Omron CX-Programmer project 新工程 (CX-Programmer 9.73)

# PLC 新PLC1: CJ1M CPU11

## Global symbols (name address type ; comment)
2000 CHANNEL  ; 打螺丝个数显示
2000.01 BOOL  ; 参数1
2000.02 BOOL  ; 参数2
2000.03 BOOL  ; DRIVER PROGRAM CH3
2000.04 BOOL  ; DRIVER PROGRAM CH4
2000.07 BOOL  ; BZ
2000.08 BOOL  ; 正常指示
2000.09 BOOL  ; 异常指示
2000.10 BOOL  ; OK
2000.11 BOOL  ; NG指示
2000.12 BOOL  ; BZ
2006.00 BOOL  ; 前A2吐油SOL
2006.02 BOOL  ; 前A1吐油SOL
2006.04 BOOL  ; A1后吐油
2006.06 BOOL  ; A2后吐油
2006.08 BOOL  ; 打油SOL
2007.00 BOOL  ; 涂布运转准备条件
2007.01 BOOL  ; MS运转准备条件
2007.06 BOOL  ; 第一步OK
2007.07 BOOL  ; 第二步OK
2007.08 BOOL  ; 第三步OK
2007.09 BOOL  ; 第四步OK
2007.11 BOOL  ; 不良
2007.12 BOOL  ; 蜂鸣器
2008.00 BOOL  ; 工件确认
2008.01 BOOL  ; 组装可信号
2008.02 BOOL  ; 完了信号
2008.03 BOOL  ; 完了信號
2008.04 BOOL  ; 报警信号
2008.05 BOOL  ; 打螺丝手柄开关
2008.08 BOOL  ; 组装回数选择
2008.09 BOOL  ; 不良解除
2008.10 BOOL  ; 消音
2008.15 BOOL  ; 运转准备ON
2014.00 BOOL  ; 前有工件传感器
2014.01 BOOL  ; 前吐油传感器
2014.02 BOOL  ; 后有工件传感器
2014.03 BOOL  ; 后吐油传感器
2014.04 BOOL  ; 后吐油开始传感器
2014.05 BOOL  ; 前吐油开始传感器
2014.06 BOOL  ; GREASE COATING CONF.2R
2014.07 BOOL  ; GREASE COATING CONF.2L
2014.08 BOOL  ; WORKPIECE CONFIEMATION
2014.09 BOOL  ; WORKPIECE SET MEMORY
2015.00 BOOL  ; 运转准备ON
2015.03 BOOL  ; 非常停止
2015.05 BOOL  ; -
2015.06 BOOL  ; 自动
2015.07 BOOL  ; 不良解除
2015.08 BOOL  ; 消音
2015.09 BOOL  ; 后涂布手动
2015.10 BOOL  ; 前涂布手动
2015.15 BOOL  ; 獶盽氨ゎ
2100.00 BOOL  ; WORKPIECE SET MEMORY
253.08 BOOL  ; CPU BATTERY LOWER
3000.00 BOOL  ; AUTO. RUN
3000.01 BOOL  ; START
3200.00 BOOL  ; PC FAULT
3200.01 BOOL  ; PATTERN FAULT
3200.02 BOOL  ; CYCLE TIME  OVER
3200.04 BOOL  ; GREASE COATING FAULT
3200.05 BOOL  ; GREASE COATING CONF. SENSOR FAULT
3201.00 BOOL  ; FAULT
3201.01 BOOL  ; ALARM RESET
3201.03 BOOL  ; FAULT RESET
3210.00 BOOL  ; RESTART PROTECTION
3210.01 BOOL  ; CONDITION OF AUTO RUN
3210.15 BOOL  ; CYCLE COMPLETE
3211.00 BOOL  ; INDIV. STEP UP
3211.04 BOOL  ; STEP UP
3211.06 BOOL  ; AUTO. RUN (DIFU)
3211.08 BOOL  ; NOT STEP MOTION
3220.00 BOOL  ; GREASE COATING START:1R
3220.01 BOOL  ; GREASE COATING GOOD:1R
3220.02 BOOL  ; GREASE COATING FAULT:1R
3221.00 BOOL  ; GREASE COATING START:1L
3221.01 BOOL  ; GREASE COATING GOOD:1L
3221.02 BOOL  ; GREASE COATING FAULT:1L
3222.00 BOOL  ; GREASE COATING START:2R
3222.01 BOOL  ; GREASE COATING GOOD:2R
3222.02 BOOL  ; GREASE COATING FAULT:2R
3223.00 BOOL  ; GREASE COATING START:2L
3223.01 BOOL  ; GREASE COATING GOOD:2L
3223.02 BOOL  ; GREASE COATING FAULT:2L
3223.08 BOOL  ; AIR SUPPLY ON
3230.00 BOOL  ; �幡R猳
3230.01 BOOL  ; GREASE COATING 1SHOT:1L
3230.02 BOOL  ; GREASE COATING 1SHOT:2R
3230.03 BOOL  ; GREASE COATING 1SHOT:2L
3240.00 BOOL  ; PATTERN FAULT
3250.00 BOOL  ; 後吐油非
3260.01 BOOL  ; spare
3260.02 BOOL  ; spare
32.00 BOOL  ; 放工件脉冲
32.01 BOOL  ; CYCLE开始
32.02 BOOL  ; NG
32.03 BOOL  ; 手动打螺丝PLS
32.04 BOOL  ; 初始化完成信号
33.00 BOOL  ; 驱动器开始控制
33.01 BOOL  ; 1st. COMPLETE BZ
33.02 BOOL  ; 2nd. COMPLETE BZ
33.03 BOOL  ; 固定过程完成
33.04 BOOL  ; 步完成蜂鸣器叫
33.05 BOOL  ; 2过程完成蜂鸣器
33.06 BOOL  ; 步完成蜂鸣器
33.07 BOOL  ; OK
33.08 BOOL  ; NG
33.09 BOOL  ; NG RESET
33.10 BOOL  ; NG
33.11 BOOL  ; BZ复位
33.12 BOOL  ; BZ
33.13 BOOL  ; 3nd. COMPLETE BZ
34.00 BOOL  ; 机种选择2
34.01 BOOL  ; 机种选择1
50.00 BOOL  ; A1后吐油
50.01 BOOL  ; 第一步后吐油完成
50.02 BOOL  ; A1前吐油
50.03 BOOL  ; 第二步前吐油完成
50.05 BOOL  ; 第三步后吐油完成
50.06 BOOL  ; A1后吐油
50.07 BOOL  ; 第四部后吐油完成
51.00 BOOL  ; 产品确认
51.02 BOOL  ; 报警
52.00 BOOL  ; A2后吐油
52.01 BOOL  ; A2后吐油
52.02 BOOL  ; A2前吐油
52.03 BOOL  ; A2前吐油
52.04 BOOL  ; A1后吐油
52.05 BOOL  ; A2后吐油
52.06 BOOL  ; A2后吐油
52.07 BOOL  ; A2后吐油
52.08 BOOL  ; A2后吐油
53.00 BOOL  ; 后吐油无工件确认
55.00 BOOL  ; 下一步吐油可以
55.01 BOOL  ; 第三步前吐油条件
58.09 BOOL  ; OK
59.00 BOOL  ; 工件正常完成
6014.00 BOOL  ; DUMMY
60.00 BOOL  ; 工件非正常移開
60.01 BOOL  ; 工件非正常移開
60.02 BOOL  ; 故障周期復位
60.03 BOOL  ; NG
60.04 BOOL  ; NG
68.00 BOOL  ; 复位OK
68.01 BOOL  ; 复位OK
80.00 BOOL  ; 自动停止PLS
80.01 BOOL  ; 一次吐油完了
80.02 BOOL  ; 吐油之後拿掉工件
80.03 BOOL  ; �R猳ok
80.04 BOOL  ; 吐油ok後拿掉工件
81.00 BOOL  ; �幡R猳
81.01 BOOL  ; 一次吐油完了
81.02 BOOL  ; 吐油之後拿掉工件
81.03 BOOL  ; �R猳ok
81.04 BOOL  ; 吐油ok後拿掉工件
82.00 BOOL  ; 手动前涂布
82.01 BOOL  ; 手动后涂布
83.00 BOOL  ; NG
83.01 BOOL  ; 蜂鸣器
90.00 BOOL  ; OK RESET START READY
90.01 BOOL  ; OK RESTART
98.00 BOOL  ; COUNTER RESET PLS
A395.11 BOOL  ; Flash MEMORY FAULT
C0118 BOOL  ; 前吐油計數
C0205 BOOL  ; 后涂布计数
D10 CHANNEL  ; 打螺丝个数
D200 CHANNEL  ; 前注油周期
D210 CHANNEL  ; 后注油周期
D220 CHANNEL  ; 注油顺序
D280 CHANNEL  ; 总生产数
H0.00 BOOL  ; Step_0丂
H0.01 BOOL  ; Step_1
H0.02 BOOL  ; Step_2
H0.03 BOOL  ; Step_3
H0.04 BOOL  ; Step_4
H0.05 BOOL  ; Step_5
H0.06 BOOL  ; Step_6
H0.07 BOOL  ; Step_7
H10 CHANNEL  ; BIT SHIFT REGISTER
H10.00 BOOL  ; 初始工作时接通
H10.01 BOOL  ; 1st. TORQUE UP
H10.02 BOOL  ; 2nd. TORQUE UP
H10.03 BOOL  ; 3rd. TORQUE UP
H1.00 BOOL  ; Step_0
H1.01 BOOL  ; Step_1
H1.02 BOOL  ; Step_2
H1.03 BOOL  ; Step_3
H1.04 BOOL  ; Step_4
T0008 BOOL  ; CYCLE TIME
T0010 BOOL  ; 自動延時
T0011 BOOL  ; INDIV. MODE
T0018 BOOL  ; OK
T0020 BOOL  ; WORKPIECE CONF. TIMER :1R
T0021 BOOL  ; WORKPIECE CONF. TIMER :1L
T0030 BOOL  ; WORKPIECE CONF. TIMER :2R
T0031 BOOL  ; WORKPIECE CONF. TIMER :2L
T0060 BOOL  ; GREASE COATING TIME:1R
T0061 BOOL  ; GREASE COATING TIME:1L
T0062 BOOL  ; GREASE COATING TIME:2R
T0063 BOOL  ; GREASE COATING TIME:2L
T0100 BOOL  ; 前有工件延时
T0101 BOOL  ; 前吐油延时
T0102 BOOL  ; 后有工件延时
T0103 BOOL  ; 后吐油延时
T0104 BOOL  ; GREASE COATING CONFIRMATION:1R
T0105 BOOL  ; GREASE COATING CONFIRMATION:1L
T0106 BOOL  ; GREASE COATING CONFIRMATION:2R
T0107 BOOL  ; GREASE COATING CONFIRMATION:2L
T0108 BOOL  ; WORKPIECE CONFIRMATION
T0109 BOOL  ; NON WORKPIECE CONFIRMATION
T0110 BOOL  ; 后吐油开始延时
T0111 BOOL  ; 前吐油开始延时
T0112 BOOL  ; 前涂布手动延时
T0113 BOOL  ; 后涂布手动延时
T0114 BOOL  ; 运转准备输入延时
T0115 BOOL  ; 自动延时
T0119 BOOL  ; 前拿掉工件后延时
T0121 BOOL  ; 后拿掉工件后延时
T0131 BOOL  ; 工件检知延时
T0132 BOOL  ; A1A2后吐油时间
T0133 BOOL  ; A1A2前吐油时间
T0135 BOOL  ; A1A2后吐油时间
T0140 BOOL  ; 工件检知无延时
T0142 BOOL  ; 工件检知无RESET
T0150 BOOL  ; A1后吐油时间
T0151 BOOL  ; A2后吐油时间
T0152 BOOL  ; A1前吐油时间
T0153 BOOL  ; A2前吐油时间
T0154 BOOL  ; A1A2后吐油时间
T0155 BOOL  ; A1吐油时间
T0156 BOOL  ; A2后吐油时间
T0157 BOOL  ; 后油油无检知工件延时
T0158 BOOL  ; A1后吐油时间
T0159 BOOL  ; A2后吐油时间
T0200 BOOL  ; 工件确认延时
T0201 BOOL  ; 工件移开时间
T0202 BOOL  ; 手动打螺丝延时
T0203 BOOL  ; 完了信号延时
T0204 BOOL  ; 驱动器开始信号延时
T0211 BOOL  ; 1st完成BZ Time
T0212 BOOL  ; 2nd完成 BZ Time
T0213 BOOL  ; 3nd完成BZTime
T0214 BOOL  ; 1固定完成时间
T0215 BOOL  ; 2固定完成时间
T0216 BOOL  ; 1固定完成时间
T0221 BOOL  ; 工件移开短延时
T0222 BOOL  ; 蜂鸣器叫时间
T0230 BOOL  ; 第1步完成响时间
T0231 BOOL  ; 第2步完成响时间
T0232 BOOL  ; 第3步完成响时间
T0233 BOOL  ; 第5步完成响时间
T0300 BOOL  ; 前A1 ON持续时间
T0301 BOOL  ; 前A2 ON开始时间
T0302 BOOL  ; 前A2 ON持续时间
T0303 BOOL  ; 前注油CYCLE结束
T0310 BOOL  ; 后A1 ON持续时间
T0311 BOOL  ; 后A2 ON开始时间
T0312 BOOL  ; 后A2 ON持续时间
T0313 BOOL  ; 后注油CYCLE结束
T10 CHANNEL  ; AUTO. MODE
T11 CHANNEL  ; INDIV. MODE
T20 CHANNEL  ; WORKPIECE CONF. TIMER :1R
T21 CHANNEL  ; WORKPIECE CONF. TIMER :1L
T30 CHANNEL  ; WORKPIECE CONF. TIMER :2R
T31 CHANNEL  ; WORKPIECE CONF. TIMER :2L
T8 CHANNEL  ; CYCLE TIME
W100.00 BOOL  ; 吐油ON开始打油
W100.01 BOOL  ; 吐油ON开始打油
W200.00 BOOL  ; 前注油 CYCLE 开始
W200.01 BOOL  ; 前A1 ON 辅助
W200.02 BOOL  ; 前A2 ON 辅助
W200.03 BOOL  ; 前吐油确认
W200.04 BOOL  ; 前吐油完成
W200.05 BOOL  ; 前A2 ON开始时间
W200.06 BOOL  ; 前注油CYCLEEND
W210.00 BOOL  ; 后注油 CYCLE 开始
W210.01 BOOL  ; 后A1 ON 辅助
W210.02 BOOL  ; 后A2 ON 辅助
W210.03 BOOL  ; 后吐油确认
W210.04 BOOL  ; 2部吐油完成
W210.05 BOOL  ; 后A2 ON开始时间
W210.06 BOOL  ; 后注油CYCLEEND
W220.00 BOOL  ; 第一步OK
W220.01 BOOL  ; 第二步OK
W220.02 BOOL  ; 第三步OK
W220.03 BOOL  ; 第四步OK
W230.00 BOOL  ; 第1步完成响一声
W231.01 BOOL  ; 第2步完成响一声
W231.02 BOOL  ; 第4步完成响一声
W231.03 BOOL  ; 第4步完成响一声
W27.04 BOOL  ; 完成蜂鸣器叫一声
W50.07 BOOL  ; 急停报警
W50.08 BOOL  ; 急停蜂鸣器
TUYOU 功能块1
后吐油 功能块1
前吐油 功能块1
吐油 功能块1
吐油1 功能块1
Further comments
1 |  | 2000.00 | c4ded7b2cadebdc0b0c42028c8bcde92f782df29 | 20
2 |  | 2000.01 | c4ded7b2cadeccdfdbb8ded7d120434831 | b2cecafd31
3 |  | 2000.02 | c4ded7b2cadeccdfdbb8ded7d120434832 | b2cecafd32
4 |  | 2000.03 | c4ded7b2cadeccdfdbb8ded7d120434833 | 4452495645522050524f4752414d20434833
5 |  | 2000.04 | c4ded7b2cadeccdfdbb8ded7d120434834 | 4452495645522050524f4752414d20434834
7 |  | 2000.08 | c4ded7b2cade90b38fed20504c | d5fdb3a3d6b8cabe
8 |  | 2000.09 | c4ded7b2cade88d98fed20504c | d2ecb3a3d6b8cabe
9 |  | 2000.10 | 90b38fed8f4997b9284f4b2920504c | 4f4b
10 |  | 2000.11 | 88d98fed8f4997b9284e472920504c | 4e47d6b8cabe
11 |  | 2000.12 | ccdebbdeb0 | 20425a
12 |  | 2006.00 | 834f838a83589368957a82508271 | c7b04132cdc2d3cd534f4c
13 |  | 2006.02 | 834f838a83589368957a8250826b | c7b04131cdc2d3cd534f4c
17 |  | 2007.00 | 895e935d8f8094f593fc82e88ff08c8f | cdbfb2bcd4cbd7aad7bcb1b8ccf5bcfe
18 |  | 2007.01 | 895e935d8f8094f593fc82e88ff08c8f | 4d53d4cbd7aad7bcb1b8ccf5bcfe
19 |  | 2007.06 | 9368957a826e826a814082518945 | b5dad2bbb2bd4f4b
20 |  | 2007.07 | 9368957a826e826a814082518db6 | b5dab6feb2bd4f4b
23 |  | 2007.11 | 88d98fed | b2bbc1bc
24 |  | 2007.12 | 83758355815b | b7e4c3f9c6f7
25 |  | 2008.00 | dcb0b88a6d9446 | b9a4bcfec8b7c8cf
26 |  | 2008.01 | bdc0b0c48ef3957489c22028c8bcde92f782df29 | d7e9d7b0bfc9d0c5bac5
30 |  | 2008.05 | 92f79574bdc0b0c420284269742d535729 | b4f2c2ddcbbfcad6b1fabfaab9d8
31 |  | 2008.08 | 92f7957489f190942032706f73914991f0 | d7e9d7b0bbd8cafdd1a1d4f1
32 |  | 2008.09 | 957397c789f08f9c5042 | b2bbc1bcbde2b3fd
33 |  | 2008.10 | b1d7b0d1d8beafc45042 | cffbd2f4
34 |  | 2008.15 | 895e935d8f8094f593fc82e88a6d9446 | d4cbd7aad7bcb1b84f4e
35 |  | 2014.00 | 838f815b834e835a836283678a6d9446825052 | c7b0d3d0b9a4bcfeb4abb8d0c6f7
36 |  | 2014.01 | 838f815b834e835a836283678a6d94468250826b | c7b0cdc2d3cdb4abb8d0c6f7
37 |  | 2014.02 | 838f817c834e835a836283678a6d94463252 | baf3d3d0b9a4bcfeb4abb8d0c6f7
38 |  | 2014.03 | 838f815b834e835a836283678a6d9446324c | baf3cdc2d3cdb4abb8d0c6f7
39 |  | 2014.04 | b8ded8bd9368957a8a6d94463152 | baf3cdc2d3cdbfaacabcb4abb8d0c6f7
40 |  | 2014.05 | b8ded8bd9368957a8a6d9446314c | c7b0cdc2d3cdbfaacabcb4abb8d0c6f7
41 |  | 2014.06 | b8ded8bd9368957a8a6d94463252 | 47524541534520434f4154494e4720434f4e462e3252
42 |  | 2014.07 | b8ded8bd9368957a8a6d9446324c | 47524541534520434f4154494e4720434f4e462e324c
43 |  | 2014.08 | dcb0b8beafc48a6d9446 | 574f524b504945434520434f4e4649454d4154494f4e
44 |  | 2014.09 | dcb0b8beafc48b4c89af | 574f524b504945434520534554204d454d4f5259
45 |  | 2015.00 | 895e935d8f8094f593fc82e8904d8d86 | d4cbd7aad7bcb1b84f4e
47 |  | 2015.05 | 8ea993ae895e935d914991f0bdb2afc196a28e679770 | 202d
48 |  | 2015.06 | 8ea993ae895e935d914991f0bdb2afc1 | d7d4b6af
49 |  | 2015.07 | 957397c789f08f9c | b2bbc1bcbde2b3fd
50 |  | 2015.08 | ccdebbdeb08fc189b9 | cffbd2f4
51 |  | 2015.09 | 9368957a312d5281405042 | baf3cdbfb2bccad6b6af
52 |  | 2015.10 | 9368957a312d4c81405042 | c7b0cdbfb2bccad6b6af
54 |  | 2100.00 | dcb0b8beafc48b4c89af | 574f524b504945434520534554204d454d4f5259
56 |  | 3000.00 | 8ea993ae895e935d9286 | 4155544f2e2052554e
57 |  | 3000.01 | 8b4e93ae8ff08c8f | 5354415254
58 |  | 3200.00 | 504388d98fed94ad90b6 | 5043204641554c54
59 |  | 3200.01 | 8370835e815b839388d98fed | 5041545445524e204641554c54
60 |  | 3200.02 | bbb2b8d9c0b2d1b5b0cadeb0 | 4359434c452054494d4520204f564552
61 |  | 3200.04 | 834f838a83589368957a88d98fed | 47524541534520434f4154494e47204641554c54
62 |  | 3200.05 | b8ded8bd9368957a835a8393835488d98fed | 47524541534520434f4154494e4720434f4e462e2053454e534f52204641554c54
63 |  | 3201.00 | 88d98fed94ad90b6 | 4641554c54
64 |  | 3201.01 | ccdebbdeb08fc189b9 | 414c41524d205245534554
65 |  | 3201.03 | 957397c789f08f9c | 4641554c54205245534554
66 |  | 3210.00 | 8dc48b4e93ae96688e7e | 524553544152542050524f54454354494f4e
67 |  | 3210.01 | 8ea993ae895e935d8ff08c8f | 434f4e444954494f4e204f46204155544f2052554e20
68 |  | 3210.15 | 31bbb2b8d98f4997b9 | 4359434c4520434f4d504c455445
69 |  | 3211.00 | 8a658cc2bdc3afccdfb1afccdf | 494e4449562e2053544550205550
70 |  | 3211.04 | bdc3afccdfb1afccdf | 53544550205550
71 |  | 3211.06 | 8ea993ae93fc82e831bcaeafc4 | 4155544f2e2052554e20284449465529
72 |  | 3211.08 | bdc3afccdf9372928682c582c882a2 | 4e4f542053544550204d4f54494f4e
73 |  | 3220.00 | 9368957a8250528a4a8e6e | 47524541534520434f4154494e472053544152543a3152
74 |  | 3220.01 | 9368957a31522d4f4b | 47524541534520434f4154494e4720474f4f443a3152
75 |  | 3220.02 | 9368957a825082712d4e47 | 47524541534520434f4154494e47204641554c543a3152
76 |  | 3221.00 | 9368957a82504c8a4a8e6e | 47524541534520434f4154494e472053544152543a314c
77 |  | 3221.01 | 9368957a314c2d4f4b | 47524541534520434f4154494e4720474f4f443a314c
78 |  | 3221.02 | 9368957a314c2d4e47 | 47524541534520434f4154494e47204641554c543a314c
79 |  | 3222.00 | 9368957a32528a4a8e6e | 47524541534520434f4154494e472053544152543a3252
80 |  | 3222.01 | 9368957a32522d4f4b | 47524541534520434f4154494e4720474f4f443a3252
81 |  | 3222.02 | 9368957a3282712d4e47 | 47524541534520434f4154494e47204641554c543a3252
82 |  | 3223.00 | 9368957a324c8a4a8e6e | 47524541534520434f4154494e472053544152543a324c
83 |  | 3223.01 | 9368957a324c2d4f4b | 47524541534520434f4154494e4720474f4f443a324c
84 |  | 3223.02 | 9368957a324c2d4e47 | 47524541534520434f4154494e47204641554c543a324c
85 |  | 3223.08 | 83478341836a8362837093ae8dec93fc82e8 | 41495220535550504c59204f4e
86 |  | 3230.00 | 9368957a3152814031bcaeafc4 | abe1a652aa6f
87 |  | 3230.01 | 9368957a314c814031bcaeafc4 | 47524541534520434f4154494e47203153484f543a314c
88 |  | 3230.02 | 9368957a3252814031bcaeafc4 | 47524541534520434f4154494e47203153484f543a3252
89 |  | 3230.03 | 9368957a324c814031bcaeafc4 | 47524541534520434f4154494e47203153484f543a324c
90 |  | 3240.00 | 8ea993ae8f878f984e47 | 5041545445524e204641554c54
94 |  | 32.00 | dcb0b8beafc4203173686f74 | b7c5b9a4bcfec2f6b3e5
95 |  | 32.01 | bbb2b8d9bdc0b0c4208a6d9446 | 4359434c45bfaacabc
96 |  | 32.02 | bbb2b8d98f4997b98a6d9446 | 4e47
97 |  | 32.03 | bdc0b0c4cadfd9bd | cad6b6afb4f2c2ddcbbf504c53
98 |  | 32.04 | 8aae97b995db8e9d | b3f5cabcbbafcdeab3c9d0c5bac5
99 |  | 33.00 | c4ded7b2cade8b4e93ae2090a78ce4 | c7fdb6afc6f7bfaacabcbfd8d6c6
100 |  | 33.01 | 825089f196da208aae97b9425a | 3173742e20434f4d504c45544520425a
101 |  | 33.02 | 3289f196da208aae97b9425a | 326e642e20434f4d504c45544520425a
102 |  | 33.03 | 92f795748d4892f6208aae97b9 | b9ccb6a8b9fdb3cccdeab3c9
103 |  | 33.04 | 92f795748d4892f6208aae97b9425a2028312f3229 | b2bdcdeab3c9b7e4c3f9c6f7bdd0
104 |  | 33.05 | 92f795748d4892f6208aae97b9425a2028322f3229 | 32b9fdb3cccdeab3c9b7e4c3f9c6f7
105 |  | 33.06 | 8dec8bc68f4997b920ccdebbdeb090a78ce4 | b2bdcdeab3c9b7e4c3f9c6f7
106 |  | 33.07 | 916795748aae97b920284f4b29 | 4f4b
108 |  | 33.09 | 957397c789f08f9cc4d8b6de | 4e47205245534554
109 |  | 33.10 | 9167957496a28aae97b920284e4729 | 4e47
110 |  | 33.11 | ccdebbdeb08fc189b995db8e9d | 425ab8b4cebb
111 |  | 33.12 | 9167957496a28aae97b920425a | 425a
112 |  | 33.13 | 3389f196da8aae97b9425a | 336e642e20434f4d504c45544520425a
138 |  | 6014.00 | 89bc90da935f | 44554d4d59
171 |  | H0.00 | bdc3afccdf30 | 537465705f308140
172 |  | H0.01 | bdc3afccdf31209368957a8250 | 537465705f3120
173 |  | H0.02 | bdc3afccdf32814088da93ae8a6d944631 | 537465705f3220
174 |  | H0.03 | bdc3afccdf338140b4b1c6afcadf93ae8dec4f6b | 537465705f33
175 |  | H0.04 | bdc3afccdf3481404e4f50 | 537465705f34
176 |  | H0.05 | bdc3afccdf3581404e4f50 | 537465705f35
177 |  | H0.06 | bdc3afccdf3681404e4f50 | 537465705f36
178 |  | H0.07 | bdc3afccdf37 | 537465705f37
179 |  | H10 | 4359434c4520424954205348494654205245474953544552 | 424954205348494654205245474953544552
180 |  | H10.00 | dcb0b8beafc48c9f8f6f | b3f5cabcb9a4d7f7cab1bdd3cda8
181 |  | H10.01 | 3189f196da20c4d9b8b1afccdf | 3173742e20544f52515545205550
182 |  | H10.02 | 3289f196da20c4d9b8b1afccdf | 326e642e20544f52515545205550
183 |  | H10.03 | 3389f196da20c4d9b8b1afccdf | 3372642e20544f52515545205550
184 |  | H1.00 | bdc3afccdf30 | 537465705f30
185 |  | H1.01 | bdc3afccdf31209368957a8251 | 537465705f3120
186 |  | H1.02 | bdc3afccdf32814088da93ae8a6d94468251 | 537465705f3220
187 |  | H1.03 | bdc3afccdf338140b4b1c6afcadf93ae8dec4f6b | 537465705f33
188 |  | H1.04 | bdc3afccdf3481404e4f50 | 537465705f34
189 |  | T0008 | bbb2b8d9c0b2d18ac48e8b | 4359434c452054494d4520
190 |  | T0010 | 8ea993ae8382815b8368 | a6dbb0caa9b5aec9
191 |  | T0011 | 8a658cc2895e935d8382815b8368 | 494e4449562e204d4f4445
193 |  | T0020 | 9368957a315288d98fed | 574f524b504945434520434f4e462e2054494d4552203a3152
194 |  | T0021 | 9368957a314c88d98fed | 574f524b504945434520434f4e462e2054494d4552203a314c
195 |  | T0030 | 9368957a325288d98fed | 574f524b504945434520434f4e462e2054494d4552203a3252
196 |  | T0031 | 9368957a325288d98fed | 574f524b504945434520434f4e462e2054494d4552203a324c
197 |  | T0060 | 9368957a8e9e8ad43152 | 47524541534520434f4154494e472054494d453a3152
198 |  | T0061 | 9368957a8e9e8ad4314c | 47524541534520434f4154494e472054494d453a314c
199 |  | T0062 | 9368957a8e9e8ad43252 | 47524541534520434f4154494e472054494d453a3252
200 |  | T0063 | 9368957a8e9e8ad4324c | 47524541534520434f4154494e472054494d453a324c
201 |  | T0100 | dcb0b8beafc48a6d94463152 | c7b0d3d0b9a4bcfed1d3cab1
202 |  | T0101 | dcb0b8beafc48a6d9446314c | c7b0cdc2d3cdd1d3cab1
203 |  | T0102 | dcb0b8beafc48a6d94463252 | baf3d3d0b9a4bcfed1d3cab1
204 |  | T0103 | dcb0b8beafc48a6d9446324c | baf3cdc2d3cdd1d3cab1
205 |  | T0104 | 9368957a31528a6d9446 | 47524541534520434f4154494e4720434f4e4649524d4154494f4e3a3152
206 |  | T0105 | 9368957a314c8a6d9446 | 47524541534520434f4154494e4720434f4e4649524d4154494f4e3a314c
207 |  | T0106 | 9368957a32528a6d9446 | 47524541534520434f4154494e4720434f4e4649524d4154494f4e3a3252
208 |  | T0107 | 9368957a324c8a6d9446 | 47524541534520434f4154494e4720434f4e4649524d4154494f4e3a324c
209 |  | T0108 | dcb0b8beafc48a6d9446 | 574f524b504945434520434f4e4649524d4154494f4e
210 |  | T0109 | dcb0b8beafc49594dcb0b896b382b58a6d9446 | 4e4f4e20574f524b504945434520434f4e4649524d4154494f4e
235 |  | T0200 | dcb0b8beafc488c092e8 | b9a4bcfec8b7c8cfd1d3cab1
236 |  | T0201 | dcb0b88ee68a4f82b58a6d9446 | b9a4bcfed2c6bfaacab1bce4
237 |  | T0202 | bdc0b0c4c0b2d0ddb8de | cad6b6afb4f2c2ddcbbfd1d3cab1
238 |  | T0203 | 8aae97b9c0b2d0ddb8de | cdeac1cbd0c5bac5d1d3cab1
240 |  | T0211 | 3189f196da8aae97b920425a8e9e8ad4 | 317374cdeab3c9425a2054696d65
241 |  | T0212 | 3289f196da8aae97b920425a8e9e8ad4 | 326e64cdeab3c920425a2054696d65
242 |  | T0213 | 3389f196da8aae97b9425a8e9e8ad4 | 336e64cdeab3c9425a54696d65
244 |  | T0215 | 92f795748aae97b920425a2d4f46468e9e8ad4 | 32b9ccb6a8cdeab3c9cab1bce4
245 |  | T0216 | 92f795748aae97b920425a8e9e8ad42028322f3229 | 31b9ccb6a8cdeab3c9cab1bce4
260 |  | T10 | 8ea993ae8382815b8368 | 4155544f2e204d4f4445
261 |  | T11 | 8a658cc2895e935d8382815b8368 | 494e4449562e204d4f4445
262 |  | T20 | 9368957a315288d98fed | 574f524b504945434520434f4e462e2054494d4552203a3152
263 |  | T21 | 9368957a314c88d98fed | 574f524b504945434520434f4e462e2054494d4552203a314c
264 |  | T30 | 9368957a325288d98fed | 574f524b504945434520434f4e462e2054494d4552203a3252
265 |  | T31 | 9368957a325288d98fed | 574f524b504945434520434f4e462e2054494d4552203a324c
266 |  | T8 | bbb2b8d9c0b2d18ac48e8b | 4359434c452054494d4520

## Program Screw_Tightening (cyclic task 0)

### Section Main
; 这个PLC程序实现了一个组装螺丝注黄油系统的控制系统。我尽可能的把注释打全了；针对OMRON的，I/O采用compobus/s通信；系统包括PLC控制器CJ1M CPU11、工件确认传感器、吐油电磁阀、打螺丝手柄开关、急停按钮、蜂鸣器等物理设备。 / 系统启动时，首先通过工件确认传感器检测工件是否到位，只有检测到工件后才会置位内部标志，并在运转准备ON置位时进入自动运行模式。若在前注油CYCLE开始或后注油CYCLE开始置位时工件确认传感器变为假，系统将暂停操作，确保工件始终在位。 / 润滑过程严格按照注油顺序执行。当注油顺序为0时，系统置位前注油CYCLE开始，驱动前A1吐油SOL和前A2吐油SOL涂润滑油，待前吐油传感器确认喷涂完成后才会递增注油顺序，只有当前步骤验证通过后才会进入下一步，避免顺序混乱。当注油顺序推进至1、2或3时，置位后注油CYCLE开始，驱动后A1吐油SOL和后A2吐油SOL完成后续喷涂，由后吐油传感器验证后继续推进流程。 / 润滑完成后，操作员按下打螺丝手柄开关触发螺丝紧固，系统根据组装回数选择执行单次或多次紧固。紧固结束后，结果通过OK指示或NG指示显示，同时更新总生产数。若T0140超时且第四步未完成，系统会置位不良标志，停止运行并激活蜂鸣器发出警报，提醒操作员处理不良品。在不良品检测或步骤完成时，蜂鸣器都会响起，确保操作员及时知晓状态。 / 为保障安全，若急停按钮被按下，系统会执行急停逻辑，关闭所有输出，防止意外发生。 / 操作员可通过不良解除恢复系统，或按消音关闭警报声。

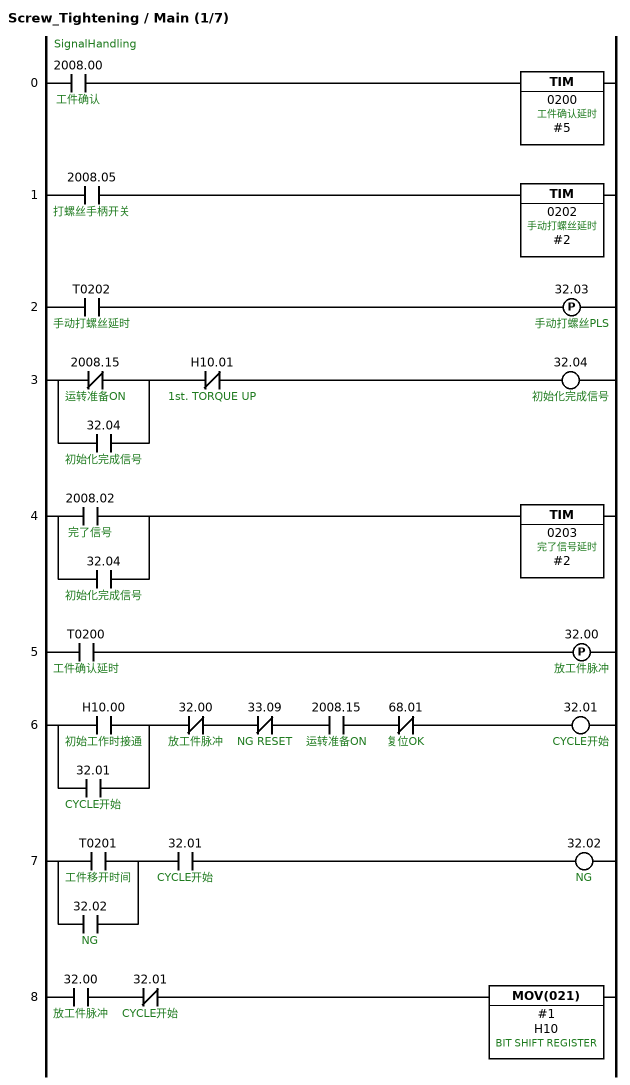
; rung 0: SignalHandling
LD 2008.00  ; 工件确认
TIM 0200 #5  ; 工件确认延时
; rung 1
LD 2008.05  ; 打螺丝手柄开关
TIM 0202 #2  ; 手动打螺丝延时
; rung 2
LD T0202  ; 手动打螺丝延时
DIFU(013) 32.03  ; 手动打螺丝PLS
; rung 3
LDNOT 2008.15  ; 运转准备ON
OR 32.04  ; 初始化完成信号
ANDNOT H10.01  ; 1st. TORQUE UP
OUT 32.04  ; 初始化完成信号
; rung 4
LD 2008.02  ; 完了信号
OR 32.04  ; 初始化完成信号
TIM 0203 #2  ; 完了信号延时
; rung 5
LD T0200  ; 工件确认延时
DIFU(013) 32.00  ; 放工件脉冲
; rung 6
LD H10.00  ; 初始工作时接通
OR 32.01  ; CYCLE开始
ANDNOT 32.00  ; 放工件脉冲
ANDNOT 33.09  ; NG RESET
AND 2008.15  ; 运转准备ON
ANDNOT 68.01  ; 复位OK
OUT 32.01  ; CYCLE开始
; rung 7
LD T0201  ; 工件移开时间
OR 32.02  ; NG
AND 32.01  ; CYCLE开始
OUT 32.02  ; NG
; rung 8
LD 32.00  ; 放工件脉冲
ANDNOT 32.01  ; CYCLE开始
MOV(021) #1 H10  ; BIT SHIFT REGISTER

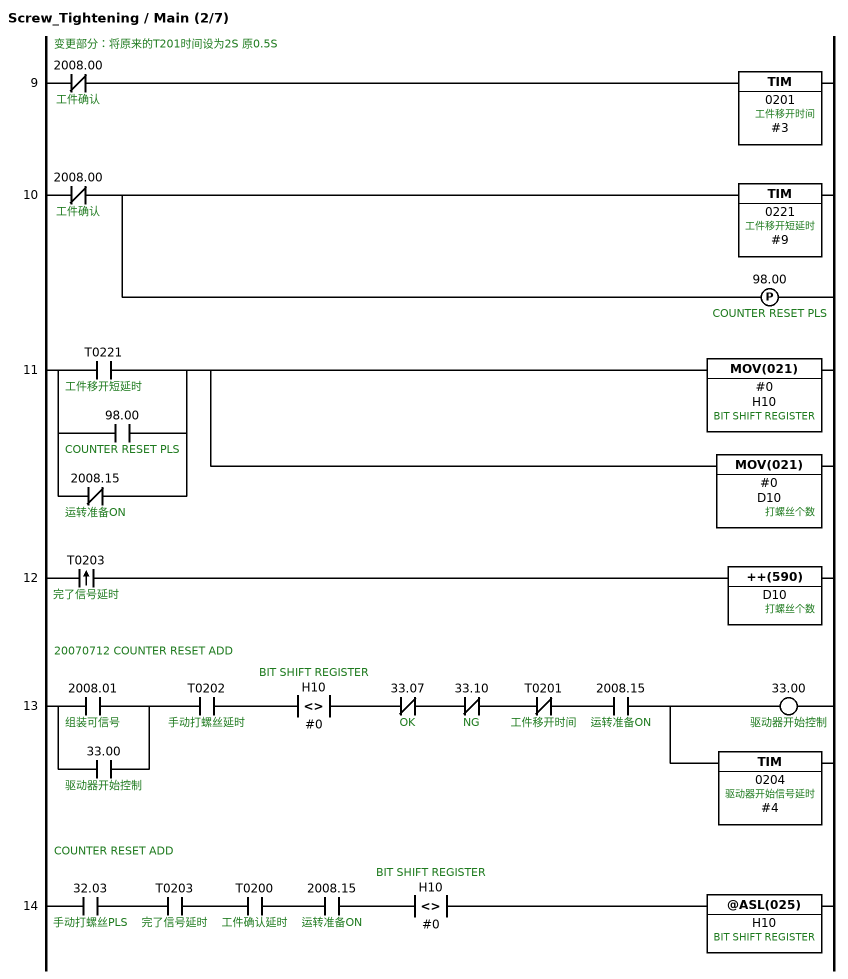
; rung 9: 变更部分：将原来的T201时间设为2S 原0.5S
LDNOT 2008.00  ; 工件确认
TIM 0201 #3  ; 工件移开时间
; rung 10
LDNOT 2008.00  ; 工件确认
TIM 0221 #9  ; 工件移开短延时
DIFU(013) 98.00  ; COUNTER RESET PLS
; rung 11
LD T0221  ; 工件移开短延时
OR 98.00  ; COUNTER RESET PLS
ORNOT 2008.15  ; 运转准备ON
MOV(021) #0 H10  ; BIT SHIFT REGISTER
MOV(021) #0 D10  ; 打螺丝个数
; rung 12
@LD T0203  ; 完了信号延时
++(590) D10  ; 打螺丝个数
; rung 13: 20070712 COUNTER RESET ADD
LD 2008.01  ; 组装可信号
OR 33.00  ; 驱动器开始控制
AND T0202  ; 手动打螺丝延时
AND<>(305) H10 #0  ; BIT SHIFT REGISTER
ANDNOT 33.07  ; OK
ANDNOT 33.10  ; NG
ANDNOT T0201  ; 工件移开时间
AND 2008.15  ; 运转准备ON
OUT 33.00  ; 驱动器开始控制
TIM 0204 #4  ; 驱动器开始信号延时
; rung 14: COUNTER RESET ADD
LD 32.03  ; 手动打螺丝PLS
AND T0203  ; 完了信号延时
AND T0200  ; 工件确认延时
AND 2008.15  ; 运转准备ON
AND<>(305) H10 #0  ; BIT SHIFT REGISTER
@ASL(025) H10  ; BIT SHIFT REGISTER

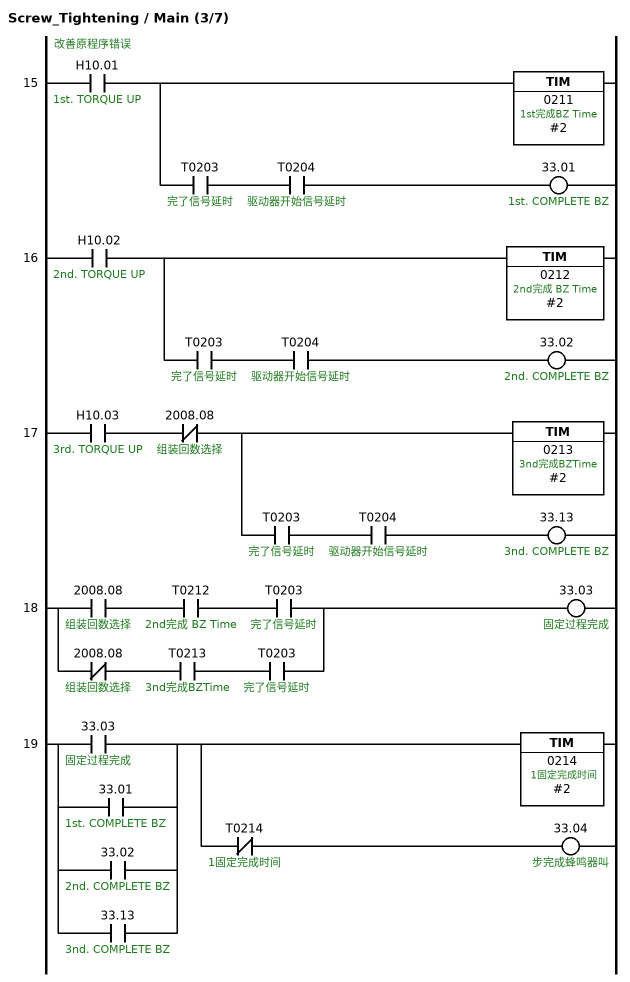
; rung 15: 改善原程序错误
LD H10.01  ; 1st. TORQUE UP
TIM 0211 #2  ; 1st完成BZ Time
AND T0203  ; 完了信号延时
AND T0204  ; 驱动器开始信号延时
OUT 33.01  ; 1st. COMPLETE BZ
; rung 16
LD H10.02  ; 2nd. TORQUE UP
TIM 0212 #2  ; 2nd完成 BZ Time
AND T0203  ; 完了信号延时
AND T0204  ; 驱动器开始信号延时
OUT 33.02  ; 2nd. COMPLETE BZ
; rung 17
LD H10.03  ; 3rd. TORQUE UP
ANDNOT 2008.08  ; 组装回数选择
TIM 0213 #2  ; 3nd完成BZTime
AND T0203  ; 完了信号延时
AND T0204  ; 驱动器开始信号延时
OUT 33.13  ; 3nd. COMPLETE BZ
; rung 18
LD 2008.08  ; 组装回数选择
AND T0212  ; 2nd完成 BZ Time
AND T0203  ; 完了信号延时
LDNOT 2008.08  ; 组装回数选择
AND T0213  ; 3nd完成BZTime
AND T0203  ; 完了信号延时
ORLD
OUT 33.03  ; 固定过程完成
; rung 19
LD 33.03  ; 固定过程完成
OR 33.01  ; 1st. COMPLETE BZ
OR 33.02  ; 2nd. COMPLETE BZ
OR 33.13  ; 3nd. COMPLETE BZ
TIM 0214 #2  ; 1固定完成时间
ANDNOT T0214  ; 1固定完成时间
OUT 33.04  ; 步完成蜂鸣器叫

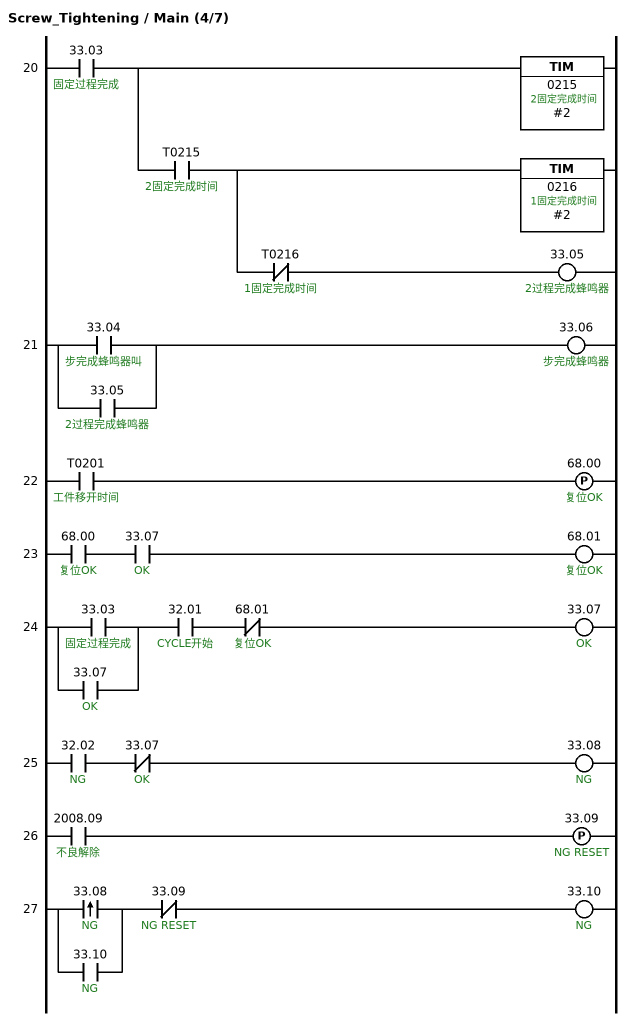
; rung 20
LD 33.03  ; 固定过程完成
TIM 0215 #2  ; 2固定完成时间
AND T0215  ; 2固定完成时间
TIM 0216 #2  ; 1固定完成时间
ANDNOT T0216  ; 1固定完成时间
OUT 33.05  ; 2过程完成蜂鸣器
; rung 21
LD 33.04  ; 步完成蜂鸣器叫
OR 33.05  ; 2过程完成蜂鸣器
OUT 33.06  ; 步完成蜂鸣器
; rung 22
LD T0201  ; 工件移开时间
DIFU(013) 68.00  ; 复位OK
; rung 23
LD 68.00  ; 复位OK
AND 33.07  ; OK
OUT 68.01  ; 复位OK
; rung 24
LD 33.03  ; 固定过程完成
OR 33.07  ; OK
AND 32.01  ; CYCLE开始
ANDNOT 68.01  ; 复位OK
OUT 33.07  ; OK
; rung 25
LD 32.02  ; NG
ANDNOT 33.07  ; OK
OUT 33.08  ; NG
; rung 26
LD 2008.09  ; 不良解除
DIFU(013) 33.09  ; NG RESET
; rung 27
@LD 33.08  ; NG
OR 33.10  ; NG
ANDNOT 33.09  ; NG RESET
OUT 33.10  ; NG

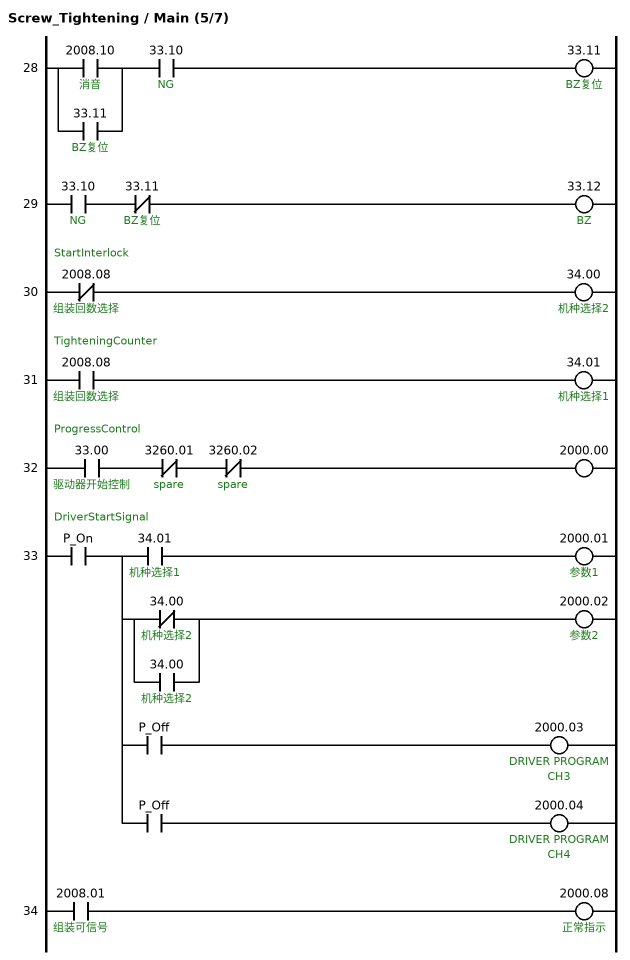
; rung 28
LD 2008.10  ; 消音
OR 33.11  ; BZ复位
AND 33.10  ; NG
OUT 33.11  ; BZ复位
; rung 29
LD 33.10  ; NG
ANDNOT 33.11  ; BZ复位
OUT 33.12  ; BZ
; rung 30: StartInterlock
LDNOT 2008.08  ; 组装回数选择
OUT 34.00  ; 机种选择2
; rung 31: TighteningCounter
LD 2008.08  ; 组装回数选择
OUT 34.01  ; 机种选择1
; rung 32: ProgressControl
LD 33.00  ; 驱动器开始控制
ANDNOT 3260.01  ; spare
ANDNOT 3260.02  ; spare
OUT 2000.00
; rung 33: DriverStartSignal
LD P_On
OUT TR0
AND 34.01  ; 机种选择1
OUT 2000.01  ; 参数1
LD TR0
LDNOT 34.00  ; 机种选择2
OR 34.00  ; 机种选择2
ANDLD
OUT 2000.02  ; 参数2
LD TR0
AND P_Off
OUT 2000.03  ; DRIVER PROGRAM CH3
LD TR0
AND P_Off
OUT 2000.04  ; DRIVER PROGRAM CH4
; rung 34
LD 2008.01  ; 组装可信号
OUT 2000.08  ; 正常指示

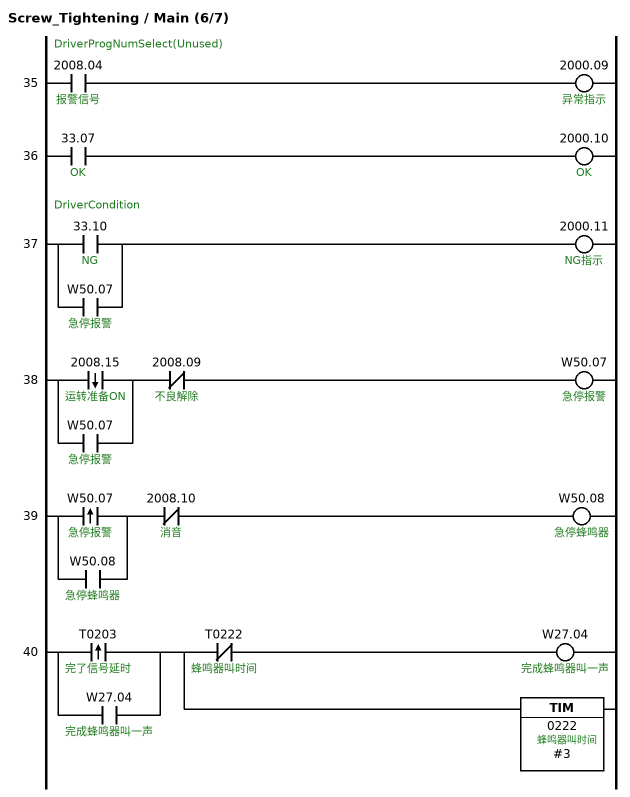
; rung 35: DriverProgNumSelect(Unused)
LD 2008.04  ; 报警信号
OUT 2000.09  ; 异常指示
; rung 36
LD 33.07  ; OK
OUT 2000.10  ; OK
; rung 37: DriverCondition
LD 33.10  ; NG
OR W50.07  ; 急停报警
OUT 2000.11  ; NG指示
; rung 38
%LD 2008.15  ; 运转准备ON
OR W50.07  ; 急停报警
ANDNOT 2008.09  ; 不良解除
OUT W50.07  ; 急停报警
; rung 39
@LD W50.07  ; 急停报警
OR W50.08  ; 急停蜂鸣器
ANDNOT 2008.10  ; 消音
OUT W50.08  ; 急停蜂鸣器
; rung 40
@LD T0203  ; 完了信号延时
OR W27.04  ; 完成蜂鸣器叫一声
OUT TR0
ANDNOT T0222  ; 蜂鸣器叫时间
OUT W27.04  ; 完成蜂鸣器叫一声
LD TR0
TIM 0222 #3  ; 蜂鸣器叫时间

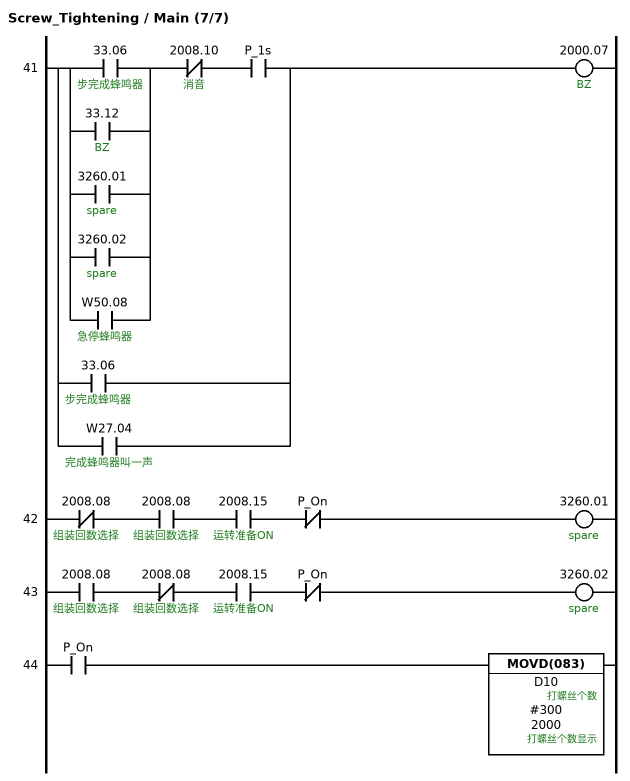
; rung 41
LD 33.06  ; 步完成蜂鸣器
OR 33.12  ; BZ
OR 3260.01  ; spare
OR 3260.02  ; spare
OR W50.08  ; 急停蜂鸣器
ANDNOT 2008.10  ; 消音
AND P_1s
LD 33.06  ; 步完成蜂鸣器
OR W27.04  ; 完成蜂鸣器叫一声
ORLD
OUT 2000.07  ; BZ
; rung 42
LDNOT 2008.08  ; 组装回数选择
AND 2008.08  ; 组装回数选择
AND 2008.15  ; 运转准备ON
ANDNOT P_On
OUT 3260.01  ; spare
; rung 43
LD 2008.08  ; 组装回数选择
ANDNOT 2008.08  ; 组装回数选择
AND 2008.15  ; 运转准备ON
ANDNOT P_On
OUT 3260.02  ; spare
; rung 44
LD P_On
MOVD(083) D10 #300 2000  ; 打螺丝个数, 打螺丝个数显示
; rung 45
END(001)

## Program GREASE_COATING (cyclic task 1)
Local symbols
R303 BOOL

### Section GREASE_COATING

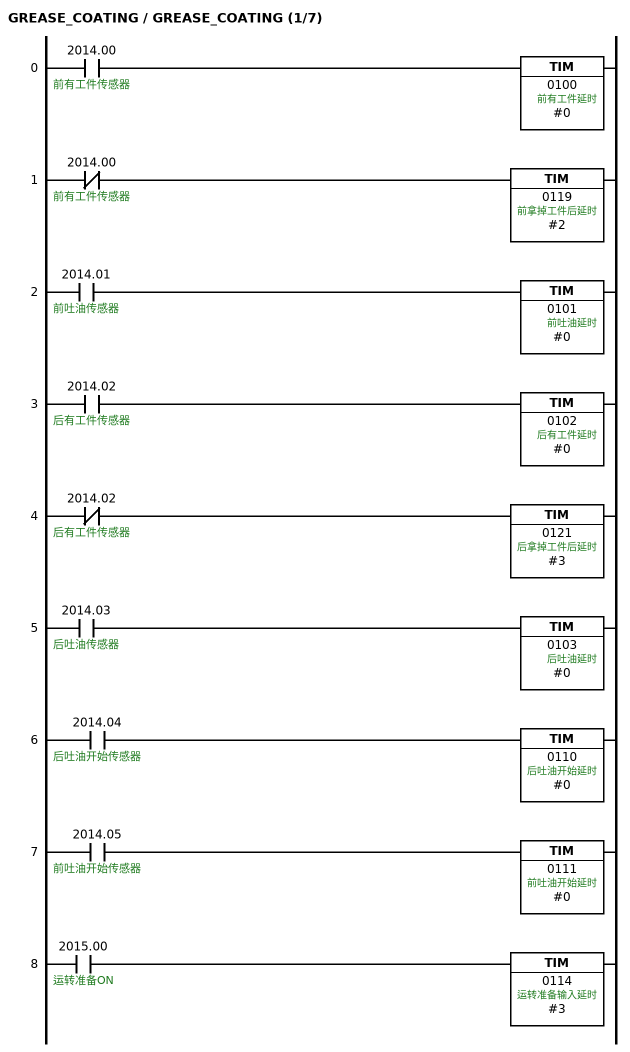
; rung 0
LD 2014.00  ; 前有工件传感器
TIM 0100 #0  ; 前有工件延时
; rung 1
LDNOT 2014.00  ; 前有工件传感器
TIM 0119 #2  ; 前拿掉工件后延时
; rung 2
LD 2014.01  ; 前吐油传感器
TIM 0101 #0  ; 前吐油延时
; rung 3
LD 2014.02  ; 后有工件传感器
TIM 0102 #0  ; 后有工件延时
; rung 4
LDNOT 2014.02  ; 后有工件传感器
TIM 0121 #3  ; 后拿掉工件后延时
; rung 5
LD 2014.03  ; 后吐油传感器
TIM 0103 #0  ; 后吐油延时
; rung 6
LD 2014.04  ; 后吐油开始传感器
TIM 0110 #0  ; 后吐油开始延时
; rung 7
LD 2014.05  ; 前吐油开始传感器
TIM 0111 #0  ; 前吐油开始延时
; rung 8
LD 2015.00  ; 运转准备ON
TIM 0114 #3  ; 运转准备输入延时

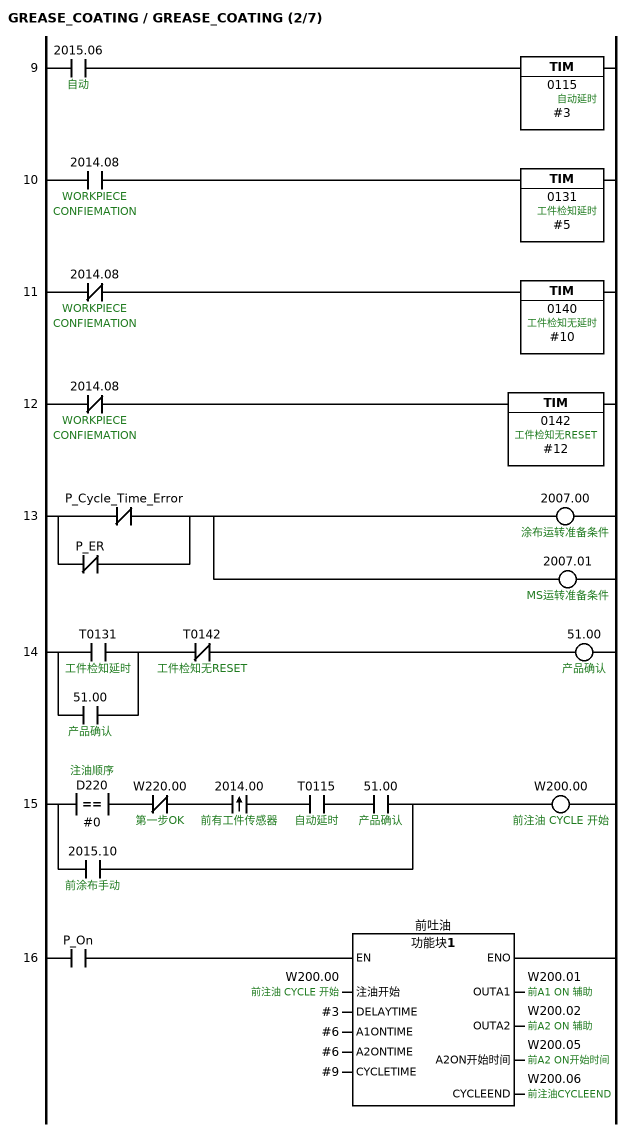
; rung 9
LD 2015.06  ; 自动
TIM 0115 #3  ; 自动延时
; rung 10
LD 2014.08  ; WORKPIECE CONFIEMATION
TIM 0131 #5  ; 工件检知延时
; rung 11
LDNOT 2014.08  ; WORKPIECE CONFIEMATION
TIM 0140 #10  ; 工件检知无延时
; rung 12
LDNOT 2014.08  ; WORKPIECE CONFIEMATION
TIM 0142 #12  ; 工件检知无RESET
; rung 13
LDNOT P_Cycle_Time_Error
ORNOT P_ER
OUT 2007.00  ; 涂布运转准备条件
OUT 2007.01  ; MS运转准备条件
; rung 14
LD T0131  ; 工件检知延时
OR 51.00  ; 产品确认
ANDNOT T0142  ; 工件检知无RESET
OUT 51.00  ; 产品确认
; rung 15
LD=(300) D220 #0  ; 注油顺序
ANDNOT W220.00  ; 第一步OK
@AND 2014.00  ; 前有工件传感器
AND T0115  ; 自动延时
AND 51.00  ; 产品确认
OR 2015.10  ; 前涂布手动
OUT W200.00  ; 前注油 CYCLE 开始
; rung 16
LD P_On
CALL 前吐油 : 功能块1 (注油开始 := W200.00, DELAYTIME := #3, A1ONTIME := #6, A2ONTIME := #6, CYCLETIME := #9, OUTA1 => W200.01, OUTA2 => W200.02, A2ON开始时间 => W200.05, CYCLEEND => W200.06)  ; 前注油 CYCLE 开始, 前A1 ON 辅助, 前A2 ON 辅助, 前A2 ON开始时间, 前注油CYCLEEND

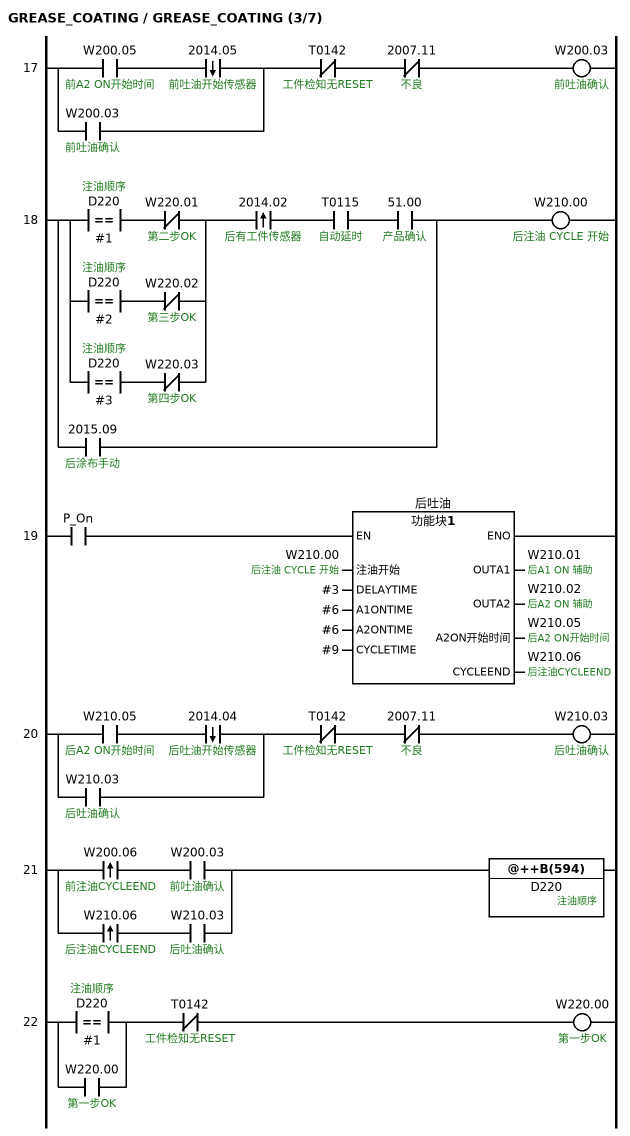
; rung 17
LD W200.05  ; 前A2 ON开始时间
%AND 2014.05  ; 前吐油开始传感器
OR W200.03  ; 前吐油确认
ANDNOT T0142  ; 工件检知无RESET
ANDNOT 2007.11  ; 不良
OUT W200.03  ; 前吐油确认
; rung 18
LD=(300) D220 #1  ; 注油顺序
ANDNOT W220.01  ; 第二步OK
LD=(300) D220 #2  ; 注油顺序
ANDNOT W220.02  ; 第三步OK
ORLD
LD=(300) D220 #3  ; 注油顺序
ANDNOT W220.03  ; 第四步OK
ORLD
@AND 2014.02  ; 后有工件传感器
AND T0115  ; 自动延时
AND 51.00  ; 产品确认
OR 2015.09  ; 后涂布手动
OUT W210.00  ; 后注油 CYCLE 开始
; rung 19
LD P_On
CALL 后吐油 : 功能块1 (注油开始 := W210.00, DELAYTIME := #3, A1ONTIME := #6, A2ONTIME := #6, CYCLETIME := #9, OUTA1 => W210.01, OUTA2 => W210.02, A2ON开始时间 => W210.05, CYCLEEND => W210.06)  ; 后注油 CYCLE 开始, 后A1 ON 辅助, 后A2 ON 辅助, 后A2 ON开始时间, 后注油CYCLEEND
; rung 20
LD W210.05  ; 后A2 ON开始时间
%AND 2014.04  ; 后吐油开始传感器
OR W210.03  ; 后吐油确认
ANDNOT T0142  ; 工件检知无RESET
ANDNOT 2007.11  ; 不良
OUT W210.03  ; 后吐油确认
; rung 21
@LD W200.06  ; 前注油CYCLEEND
AND W200.03  ; 前吐油确认
@LD W210.06  ; 后注油CYCLEEND
AND W210.03  ; 后吐油确认
ORLD
@++B(594) D220  ; 注油顺序
; rung 22
LD=(300) D220 #1  ; 注油顺序
OR W220.00  ; 第一步OK
ANDNOT T0142  ; 工件检知无RESET
OUT W220.00  ; 第一步OK

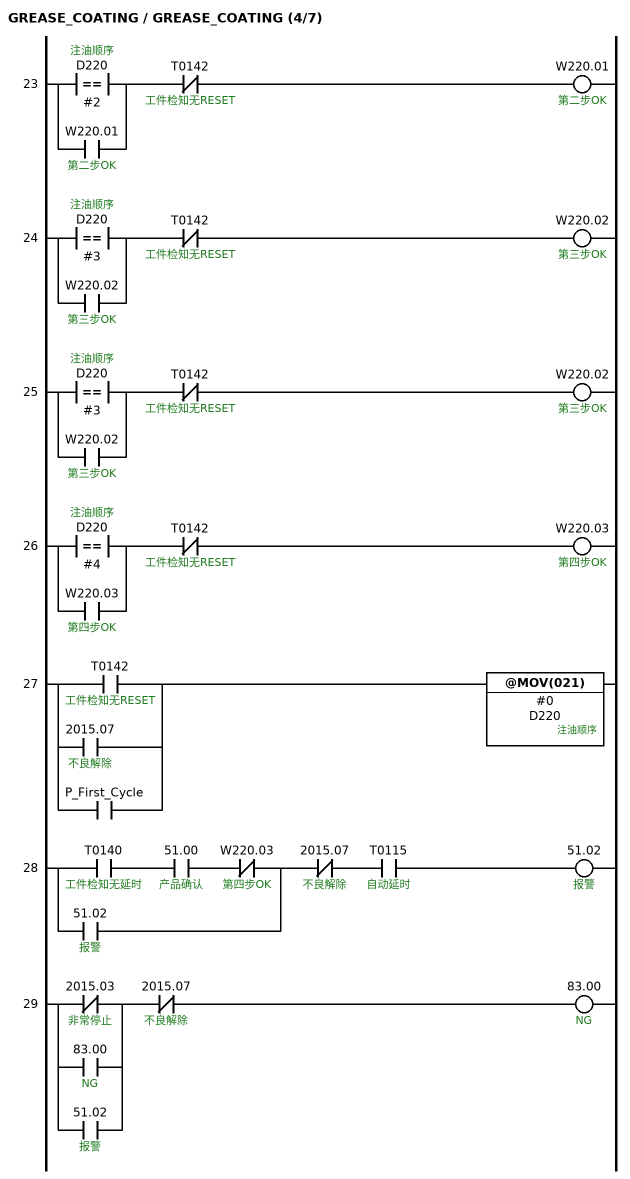
; rung 23
LD=(300) D220 #2  ; 注油顺序
OR W220.01  ; 第二步OK
ANDNOT T0142  ; 工件检知无RESET
OUT W220.01  ; 第二步OK
; rung 24
LD=(300) D220 #3  ; 注油顺序
OR W220.02  ; 第三步OK
ANDNOT T0142  ; 工件检知无RESET
OUT W220.02  ; 第三步OK
; rung 25
LD=(300) D220 #3  ; 注油顺序
OR W220.02  ; 第三步OK
ANDNOT T0142  ; 工件检知无RESET
OUT W220.02  ; 第三步OK
; rung 26
LD=(300) D220 #4  ; 注油顺序
OR W220.03  ; 第四步OK
ANDNOT T0142  ; 工件检知无RESET
OUT W220.03  ; 第四步OK
; rung 27
LD T0142  ; 工件检知无RESET
OR 2015.07  ; 不良解除
OR P_First_Cycle
@MOV(021) #0 D220  ; 注油顺序
; rung 28
LD T0140  ; 工件检知无延时
AND 51.00  ; 产品确认
ANDNOT W220.03  ; 第四步OK
OR 51.02  ; 报警
ANDNOT 2015.07  ; 不良解除
AND T0115  ; 自动延时
OUT 51.02  ; 报警
; rung 29
LDNOT 2015.03  ; 非常停止
OR 83.00  ; NG
OR 51.02  ; 报警
ANDNOT 2015.07  ; 不良解除
OUT 83.00  ; NG

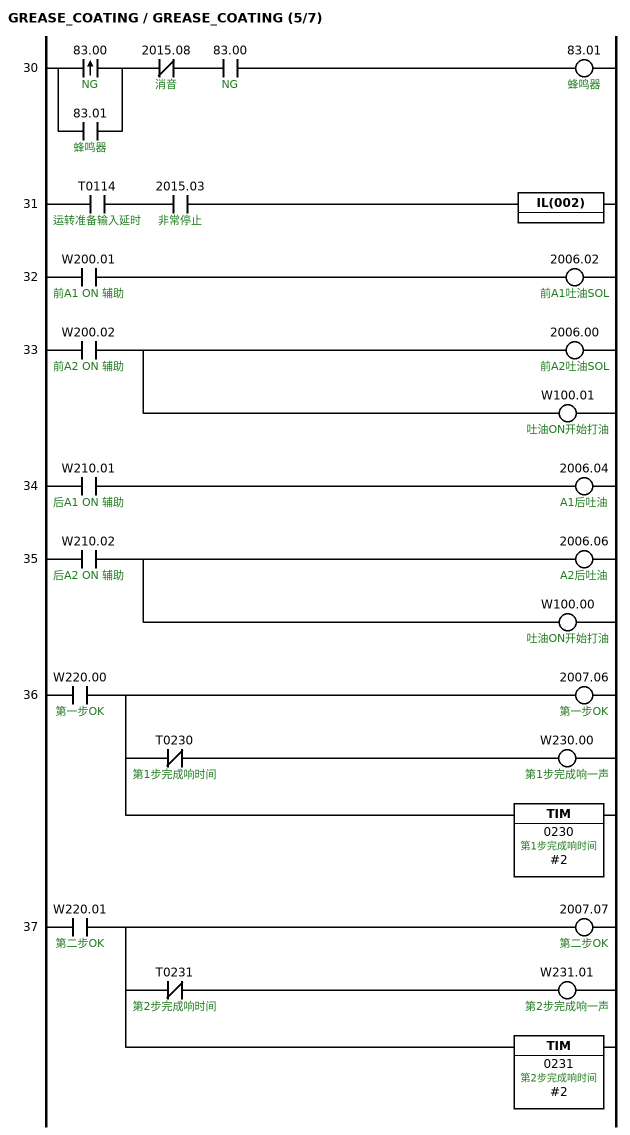
; rung 30
@LD 83.00  ; NG
OR 83.01  ; 蜂鸣器
ANDNOT 2015.08  ; 消音
AND 83.00  ; NG
OUT 83.01  ; 蜂鸣器
; rung 31
LD T0114  ; 运转准备输入延时
AND 2015.03  ; 非常停止
IL(002)
; rung 32
LD W200.01  ; 前A1 ON 辅助
OUT 2006.02  ; 前A1吐油SOL
; rung 33
LD W200.02  ; 前A2 ON 辅助
OUT 2006.00  ; 前A2吐油SOL
OUT W100.01  ; 吐油ON开始打油
; rung 34
LD W210.01  ; 后A1 ON 辅助
OUT 2006.04  ; A1后吐油
; rung 35
LD W210.02  ; 后A2 ON 辅助
OUT 2006.06  ; A2后吐油
OUT W100.00  ; 吐油ON开始打油
; rung 36
LD W220.00  ; 第一步OK
OUT TR0
OUT 2007.06  ; 第一步OK
ANDNOT T0230  ; 第1步完成响时间
OUT W230.00  ; 第1步完成响一声
LD TR0
TIM 0230 #2  ; 第1步完成响时间
; rung 37
LD W220.01  ; 第二步OK
OUT TR0
OUT 2007.07  ; 第二步OK
ANDNOT T0231  ; 第2步完成响时间
OUT W231.01  ; 第2步完成响一声
LD TR0
TIM 0231 #2  ; 第2步完成响时间

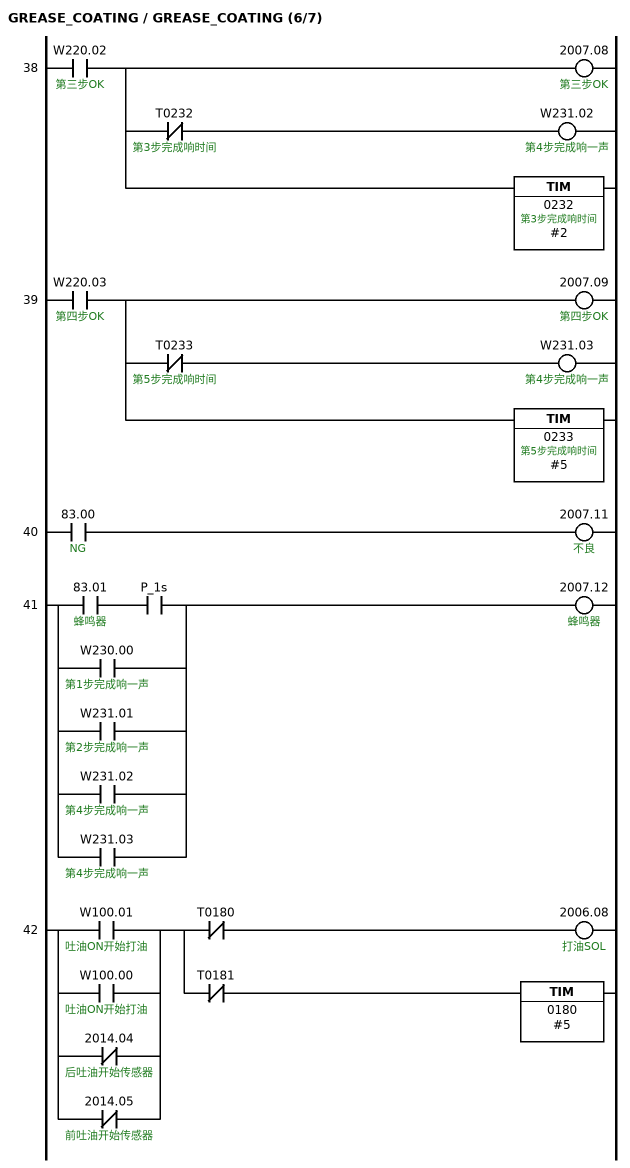
; rung 38
LD W220.02  ; 第三步OK
OUT TR0
OUT 2007.08  ; 第三步OK
ANDNOT T0232  ; 第3步完成响时间
OUT W231.02  ; 第4步完成响一声
LD TR0
TIM 0232 #2  ; 第3步完成响时间
; rung 39
LD W220.03  ; 第四步OK
OUT TR0
OUT 2007.09  ; 第四步OK
ANDNOT T0233  ; 第5步完成响时间
OUT W231.03  ; 第4步完成响一声
LD TR0
TIM 0233 #5  ; 第5步完成响时间
; rung 40
LD 83.00  ; NG
OUT 2007.11  ; 不良
; rung 41
LD 83.01  ; 蜂鸣器
AND P_1s
OR W230.00  ; 第1步完成响一声
OR W231.01  ; 第2步完成响一声
OR W231.02  ; 第4步完成响一声
OR W231.03  ; 第4步完成响一声
OUT 2007.12  ; 蜂鸣器
; rung 42
LD W100.01  ; 吐油ON开始打油
OR W100.00  ; 吐油ON开始打油
ORNOT 2014.04  ; 后吐油开始传感器
ORNOT 2014.05  ; 前吐油开始传感器
OUT TR0
ANDNOT T0180
OUT 2006.08  ; 打油SOL
LD TR0
ANDNOT T0181
TIM 0180 #5

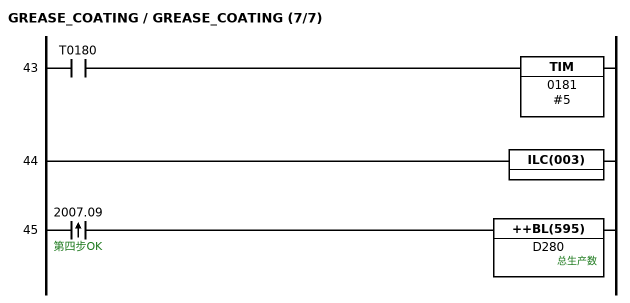
; rung 43
LD T0180
TIM 0181 #5
; rung 44
ILC(003)
; rung 45
@LD 2007.09  ; 第四步OK
++BL(595) D280  ; 总生产数
; rung 46
END(001)

### Section END
; rung 0
END(001)

## Function block 功能块1
VAR_INPUT
  注油开始 : BOOL;
  DELAYTIME : WORD;
  A1ONTIME : WORD;
  A2ONTIME : WORD;
  CYCLETIME : WORD;
END_VAR
VAR_OUTPUT
  OUTA1 : BOOL;
  OUTA2 : BOOL;
  A2ON开始时间 : BOOL;
  CYCLEEND : BOOL;
END_VAR
VAR
  CYCLESTART : BOOL;
  SOL1 : TIMER;
  DELAY1 : TIMER;
  CYCLE1 : TIMER;
  SOL2 : TIMER;
END_VAR

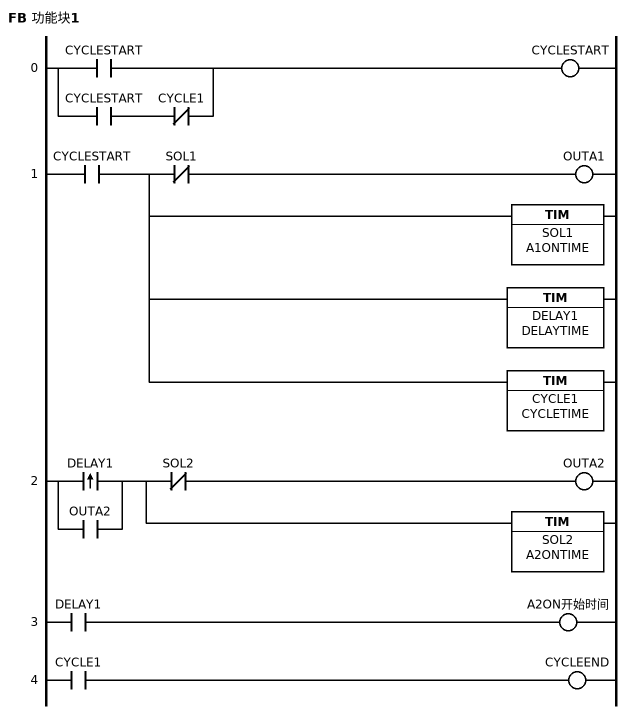
; rung 0
LD CYCLESTART
LD CYCLESTART
ANDNOT CYCLE1
ORLD
OUT CYCLESTART
; rung 1
LD CYCLESTART
OUT TR0
ANDNOT SOL1
OUT OUTA1
LD TR0
TIM SOL1 A1ONTIME
TIM DELAY1 DELAYTIME
TIM CYCLE1 CYCLETIME
; rung 2
@LD DELAY1
OR OUTA2
OUT TR0
ANDNOT SOL2
OUT OUTA2
LD TR0
TIM SOL2 A2ONTIME
; rung 3
LD DELAY1
OUT A2ON开始时间
; rung 4
LD CYCLE1
OUT CYCLEEND